Staubli VAL3: parseMovement.pgx

program parseMovement()
begin
  putln(sInput)
end
